// TIA Portal V16 export
// export: Created 2021-07-12T14:47:17.3709134Z, ExportSetting WithDefaults, DisplayName Totally Integrated Automation Portal, DisplayVersion V16, DisplayName TIA Portal Version Control Interface, DisplayVersion V16, DisplayName TIA Portal Openness, DisplayVersion V16, DisplayName STEP 7 Professional, DisplayVersion V16, DisplayName STEP 7 Safety, DisplayVersion V16, DisplayName WinCC Professional, DisplayVersion V16
DATA_BLOCK "SimaHydTO_AxisAdvanced_PosAxis_DB_1"   // DB9
FAMILY : SimaHydTO/LAxisBasics
VERSION : 1.0
// stored: AutoNumber true, DBAccessibleFromOPCUA true, InstanceOfName SimaHydTO_AxisAdvanced_PosAxis, InstanceOfType FB
"SimaHydTO_AxisAdvanced_PosAxis"
   // VAR_INPUT
   //    axis : TO_PositioningAxis;
   //    moveRelativeExecute : Bool;
   //    moveRelativeDistance : LReal;
   //    moveAbsoluteExecute : Bool;
   //    moveAbsolutePosition : LReal;
   //    moveAbsoluteDirection : Int;
   //    moveAbsPositionControlled : Bool;
   //    haltExecute : Bool;
   //    haltAbortAcceleration : Bool;
   //    Velocity : LReal;
   //    Acceleration : LReal;
   //    Deceleration : LReal;
   //    Jerk : LReal;
   // END_VAR
   // VAR_OUTPUT
   //    moveRelativeDone { ExternalWritable := 'False'} : Bool;
   //    moveRelativeBusy { ExternalWritable := 'False'} : Bool;
   //    moveAbsoluteDone { ExternalWritable := 'False'} : Bool;
   //    moveAbsoluteBusy { ExternalWritable := 'False'} : Bool;
   //    haltDone { ExternalWritable := 'False'} : Bool;
   //    haltBusy { ExternalWritable := 'False'} : Bool;
   //    commandAborted { ExternalWritable := 'False'} : Bool;
   //    error { ExternalWritable := 'False'} : Bool;
   //    errorID { ExternalWritable := 'False'} : Word;
   //    statusID { ExternalWritable := 'False'} : Int;
   // END_VAR
   // VAR
   //    instMcMoveRelative { ExternalAccessible := 'False'; ExternalVisible := 'False'; ExternalWritable := 'False'; S7_SetPoint := 'True'} : MC_MOVERELATIVE;
   //    instMcMoveAbsolute { ExternalAccessible := 'False'; ExternalVisible := 'False'; ExternalWritable := 'False'; S7_SetPoint := 'True'} : MC_MOVEABSOLUTE;
   //    instMcHalt { ExternalAccessible := 'False'; ExternalVisible := 'False'; ExternalWritable := 'False'; S7_SetPoint := 'True'} : MC_HALT;
   //    statCommandAborted { ExternalAccessible := 'False'; ExternalVisible := 'False'; ExternalWritable := 'False'} : Array[1..32] of Bool;
   //    statError { ExternalAccessible := 'False'; ExternalVisible := 'False'; ExternalWritable := 'False'} : Array[1..32] of Bool;
   //    statErrorID { ExternalAccessible := 'False'; ExternalVisible := 'False'; ExternalWritable := 'False'} : Array[1..32] of Word;
   //    instMoveAbsOpenLoop { S7_SetPoint := 'True'} : "LSimaHydTO_MC_MoveAbsOpenLoop";
   // END_VAR
BEGIN
END_DATA_BLOCK
